# EPICS substitutions: examplesTop/ndsex1App/Db/StateMachine.substitutions
file "nds3_StateMachine.template" {
pattern
{
    BOARDTYPE,
    BOARDTYPEIDX,
    CBS1,
    CBS2,
    STATEMACHINE_PARENT,
    STATEMACHINE_NAME,
}

{
    "B",
    "0",
    "TEST",
    "FCT0",
    "",
    "StateMachine",
}

}
